Fanuc KAREL source: ko00086.KL

-- PROVISIONAL review KL for V1013-1; original PC SHA256 f61f0a01a250e113213a1465e3ed01dacbe04bff2d2815313862158f4bf36185
-- Incomplete behavior may be omitted. Consult companion uncertainty JSON. Do not deploy.
PROGRAM KO00086
%NOLOCKGROUP
BEGIN
  -- UNRESOLVED_PC offsets 5-12; opcodes 9D,23
  -- UNRESOLVED_PC offsets 17-69; opcodes 27,27,49,7E,AD,27,49,7E,AD,22,31,7E,4A
  -- UNRESOLVED_PC offsets 74-78; opcodes 7F
END KO00086
